Fanuc KAREL source: webkeep.kl

PROGRAM webkeep
%COMMENT = 'v2'
%NOLOCKGROUP
%NOPAUSE=ERROR+COMMAND+TPENABLE
%NOBUSYLAMP

CONST

	R_WEBKEEP = 42

VAR

	STATUS: INTEGER
	return_code: INTEGER

BEGIN

	SET_REAL_REG(R_WEBKEEP, 0, STATUS)
	return_code = 204

END webkeep
